FUNCTION_BLOCK AI_Temperature_Channel IMPLEMENTS I_AI_Temperature, I_AI_percentage
VAR_INPUT
	terminal_address		: WORD;
	CoE_communication_handler	: I_CoE_communication_handler;
END_VAR
VAR_OUTPUT
END_VAR
VAR
	_adc_min        : INT;
    _adc_max        : INT;
	_physical_min 	: INT;
	_physical_max 	: INT;
	_channel_number : UINT;
	_rValue			: REAL;
	_wcState		: BOOL;
	
	// ===============================================================================
	// CoE handling  
    // ==============
    _CoE_prop_handler      : CoE_property_handler;
    _CoE_channel_offset     : INT;
    index_1 				: WORD:= 16#8000 + INT_TO_WORD(_CoE_channel_offset);	
    // ====  CoE properties  ===========
	_p_Enable_user_scale    		: CoE_property(Index:=index_1 , SubIndex:=1, PropertyType:=Tc2_Utilities.ARGTYPE_BOOL, writable:=TRUE, propertyType:=0, pollingInterval:=T#5S);
	_p_Presentation 				: CoE_property(Index:=index_1 , SubIndex:=2, PropertyType:=Tc2_Utilities.ARGTYPE_USINT, writable:=TRUE, propertyType:=0, pollingInterval:=T#5S);			// DT0800EN03
	_p_Watchdog 					: CoE_property(Index:=index_1 , SubIndex:=5, PropertyType:=Tc2_Utilities.ARGTYPE_USINT, writable:=TRUE, propertyType:=0, pollingInterval:=T#5S);			// DT0801EN02
	_p_Enable_user_calibration  	: CoE_property(Index:=index_1 , SubIndex:=7, PropertyType:=Tc2_Utilities.ARGTYPE_BOOL, writable:=TRUE, propertyType:=0, pollingInterval:=T#5S);
	_p_Enable_vendor_calibration    : CoE_property(Index:=index_1 , SubIndex:=8, PropertyType:=Tc2_Utilities.ARGTYPE_BOOL, writable:=TRUE, propertyType:=0, pollingInterval:=T#5S);
	_p_Offset   					: CoE_property(Index:=index_1 , SubIndex:=17, PropertyType:=Tc2_Utilities.ARGTYPE_INT, writable:=TRUE, propertyType:=0, pollingInterval:=T#5S);
	_p_Gain 						: CoE_property(Index:=index_1 , SubIndex:=18, PropertyType:=Tc2_Utilities.ARGTYPE_DINT, writable:=TRUE, propertyType:=0, pollingInterval:=T#5S);
	_p_Default_output   			: CoE_property(Index:=index_1 , SubIndex:=19, PropertyType:=Tc2_Utilities.ARGTYPE_INT, writable:=TRUE, propertyType:=0, pollingInterval:=T#5S);
	_p_Default_output_ramp  		: CoE_property(Index:=index_1 , SubIndex:=20, PropertyType:=Tc2_Utilities.ARGTYPE_UINT, writable:=TRUE, propertyType:=0, pollingInterval:=T#5S);
	_p_User_calibration_offset  	: CoE_property(Index:=index_1 , SubIndex:=21, PropertyType:=Tc2_Utilities.ARGTYPE_INT, writable:=TRUE, propertyType:=0, pollingInterval:=T#5S);
	_p_User_calibration_gain    	: CoE_property(Index:=index_1 , SubIndex:=22, PropertyType:=Tc2_Utilities.ARGTYPE_UINT, writable:=TRUE, propertyType:=0, pollingInterval:=T#5S);
	// ==============
	_properties  : ARRAY[1..11]OF I_CoE_property:=[
		_p_Enable_user_scale, _p_Presentation, _p_Watchdog, _p_Enable_user_calibration, _p_Enable_vendor_calibration, _p_Offset,
		_p_Gain, _p_Default_output, _p_Default_output_ramp, _p_User_calibration_offset, _p_User_calibration_gain];
	// ===============================================================================
    
	
	//  ====  I_AI_percentage  ====
	_max_value 	: REAL:=10.0;
	_min_value 	: REAL:=0.0;
	_value: REAL;
	
	_errId: HAL_ErrorEnum;
    neg_wcState: f_trig;
END_VAR

// CoE Property handling 
_CoE_prop_handler(terminal_address:=terminal_address, CoE_communication_handler:=CoE_communication_handler, CoE_properties:=_properties);

neg_wcState(CLK:=_wcState);
IF neg_wcState.Q THEN
    ;
END_IF

PROPERTY errId : HAL_ErrorEnum
GET
errId := _errId;
END_GET
END_PROPERTY

METHOD FB_init : BOOL
VAR_INPUT
	bInitRetains 	: BOOL; // if TRUE, the retain variables are initialized (warm start / cold start)
	bInCopyCode 	: BOOL;  // if TRUE, the instance afterwards gets moved into the copy code (online change)
    adc_min         : INT;
    adc_max         : INT;
	physical_min 	: INT;
	physical_max 	: INT;
	channel_number  : UINT;
END_VAR

VAR
	i: UINT;
END_VAR

_adc_min        := adc_min;
_adc_max        := adc_max;
_physical_min 	:= physical_min;
_physical_max 	:= physical_max;
_channel_number :=channel_number;

CASE channel_number OF
	1:
		_CoE_channel_offset:=16#0;
	2:
		_CoE_channel_offset:=16#10;
	3:
		_CoE_channel_offset:=16#20;
	4:
		_CoE_channel_offset:=16#30;
END_CASE
END_METHOD

METHOD get_Default_output : BOOL
VAR
    targ_value : Tc2_Utilities.T_Arg;
END_VAR
VAR_OUTPUT
	value	: INT;
END_VAR
get_Default_output:=_p_Default_output.get_value(value=>targ_value, errId => );
IF get_Default_output THEN
    MEMCPY(ADR(value), targ_value.pData, targ_value.cbLen);
END_IF
END_METHOD

METHOD get_Default_output_ramp : BOOL
VAR
    targ_value : Tc2_Utilities.T_Arg;
END_VAR
VAR_OUTPUT
	value	: UINT;
END_VAR
get_Default_output_ramp:=_p_Default_output_ramp.get_value(value=>targ_value, errId => );
IF get_Default_output_ramp THEN
    MEMCPY(ADR(value), targ_value.pData, targ_value.cbLen);
END_IF
END_METHOD

METHOD get_Enable_user_calibration : BOOL
VAR
    targ_value : Tc2_Utilities.T_Arg;
END_VAR
VAR_OUTPUT
	value	: BOOL;
END_VAR
get_Enable_user_calibration:=_p_Enable_user_calibration.get_value(value=>targ_value, errId => );
IF get_Enable_user_calibration THEN
    MEMCPY(ADR(value), targ_value.pData, targ_value.cbLen);
END_IF
END_METHOD

METHOD get_Enable_user_scale : BOOL
VAR
    targ_value : Tc2_Utilities.T_Arg;
END_VAR
VAR_OUTPUT
	value	: BOOL;
END_VAR
get_Enable_user_scale:=_p_Enable_user_scale.get_value(value=>targ_value, errId => );
IF get_Enable_user_scale THEN
    MEMCPY(ADR(value), targ_value.pData, targ_value.cbLen);
END_IF
END_METHOD

METHOD get_Enable_vendor_calibration : BOOL
VAR
    targ_value : Tc2_Utilities.T_Arg;
END_VAR
VAR_OUTPUT
	value	: BOOL;
END_VAR
get_Enable_vendor_calibration:=_p_Enable_vendor_calibration.get_value(value=>targ_value, errId => );
IF get_Enable_vendor_calibration THEN
    MEMCPY(ADR(value), targ_value.pData, targ_value.cbLen);
END_IF
END_METHOD

METHOD get_Gain : BOOL
VAR
    targ_value : Tc2_Utilities.T_Arg;
END_VAR
VAR_OUTPUT
	value	: DINT;
END_VAR
get_Gain:=_p_Gain.get_value(value=>targ_value, errId => );
IF get_Gain THEN
    MEMCPY(ADR(value), targ_value.pData, targ_value.cbLen);
END_IF
END_METHOD

METHOD get_Offset : BOOL
VAR
    targ_value : Tc2_Utilities.T_Arg;
END_VAR
VAR_OUTPUT
	value	: INT;
END_VAR
get_Offset:=_p_Offset.get_value(value=>targ_value, errId => );
IF get_Offset THEN
    MEMCPY(ADR(value), targ_value.pData, targ_value.cbLen);
END_IF
END_METHOD

METHOD get_Presentation : BOOL
VAR
	usint_value: USINT;
    targ_value : Tc2_Utilities.T_Arg;
END_VAR
VAR_OUTPUT
	value	: ENU_DT0801EN03;
END_VAR
get_Presentation:=_p_Presentation.get_value(value=>targ_value, errId => );
IF get_Presentation THEN
    MEMCPY(ADR(usint_value), targ_value.pData, targ_value.cbLen);
    value:=USINT_TO_INT(usint_value);
END_IF
END_METHOD

METHOD get_User_calibration_gain : BOOL
VAR
    targ_value : Tc2_Utilities.T_Arg;
END_VAR
VAR_OUTPUT
	value	: UINT;
END_VAR
get_User_calibration_gain:=_p_User_calibration_gain.get_value(value=>targ_value, errId => );
IF get_User_calibration_gain THEN
    MEMCPY(ADR(value), targ_value.pData, targ_value.cbLen);
END_IF
END_METHOD

METHOD get_User_calibration_offset : BOOL
VAR
    targ_value : Tc2_Utilities.T_Arg;
END_VAR
VAR_OUTPUT
	value	: INT;
END_VAR
get_User_calibration_offset:=_p_User_calibration_offset.get_value(value=>targ_value, errId => );
IF get_User_calibration_offset THEN
    MEMCPY(ADR(value), targ_value.pData, targ_value.cbLen);
END_IF
END_METHOD

METHOD get_Watchdog : BOOL
VAR
	usint_value: USINT;
    targ_value : Tc2_Utilities.T_Arg;
END_VAR
VAR_OUTPUT
	value	: ENU_DT0800EN02;
END_VAR
get_Watchdog:=_p_Watchdog.get_value(value=>targ_value, errId => );
IF get_Watchdog THEN
    MEMCPY(ADR(usint_value), targ_value.pData, targ_value.cbLen);
    value:=USINT_TO_INT(usint_value);
END_IF
END_METHOD

PROPERTY io_status_Error : bool
GET
END_GET
SET
END_SET
END_PROPERTY

PROPERTY io_status_Limit_1_greater_value : bool
GET
END_GET
SET
END_SET
END_PROPERTY

PROPERTY io_status_Limit_1_smaller_value : bool
GET
END_GET
SET
END_SET
END_PROPERTY

PROPERTY io_status_Limit_2_greater_value : bool
GET
END_GET
SET
END_SET
END_PROPERTY

PROPERTY io_status_Limit_2_smaller_value : bool
GET
END_GET
SET
END_SET
END_PROPERTY

PROPERTY io_status_Overrange : bool
GET
END_GET
SET
END_SET
END_PROPERTY

PROPERTY io_status_Sync_error : bool
GET
END_GET
SET
END_SET
END_PROPERTY

PROPERTY io_status_TxPDO_State : bool
GET
END_GET
SET
END_SET
END_PROPERTY

PROPERTY io_status_TxPDO_Toggle : bool
GET
END_GET
SET
END_SET
END_PROPERTY

PROPERTY io_status_Underrange : bool
GET
END_GET
SET
END_SET
END_PROPERTY

PROPERTY max_value : REAL
GET
max_value := _max_value;
END_GET
SET
IF max_value <= 0 THEN
	_max_value := 0.0001;
ELSE
	_max_value := max_value;
END_IF
END_SET
END_PROPERTY

PROPERTY min_value : REAL
GET
min_value := _min_value;
END_GET
SET
_min_value := min_value;
END_SET
END_PROPERTY

PROPERTY rValue : REAL
GET
rValue:=_rValue;
END_GET
SET
IF rValue < DINT_TO_REAL(_physical_min) THEN
	_errId := 6;
ELSIF rValue > DINT_TO_REAL(_physical_max) THEN
	_errId := 7;
ELSE
	_rValue := rValue;
END_IF
END_SET
END_PROPERTY

METHOD set_Default_output : BOOL
VAR_INPUT
	value	: INT;
END_VAR
set_Default_output:=_p_Default_output.set_value(value:=Tc2_Utilities.F_INT(in:=value));
END_METHOD

METHOD set_Default_output_ramp : BOOL
VAR_INPUT
	value	: UINT;
END_VAR
set_Default_output_ramp:=_p_Default_output_ramp.set_value(value:=Tc2_Utilities.F_UINT(in:=value));
END_METHOD

METHOD set_Enable_user_calibration : BOOL
VAR_INPUT
	value	: BOOL;
END_VAR
set_Enable_user_calibration:=_p_Enable_user_calibration.set_value(value:=Tc2_Utilities.F_BOOL(in:=value));
END_METHOD

METHOD set_Enable_user_scale : BOOL
VAR_INPUT
	value	: BOOL;
END_VAR
set_Enable_user_scale:=_p_Enable_user_scale.set_value(value:=Tc2_Utilities.F_BOOL(in:=value));
END_METHOD

METHOD set_Enable_vendor_calibration : BOOL
VAR_INPUT
	value	: BOOL;
END_VAR
set_Enable_vendor_calibration:=_p_Enable_vendor_calibration.set_value(value:=Tc2_Utilities.F_BOOL(in:=value));
END_METHOD

METHOD set_Gain : BOOL
VAR_INPUT
	value	: DINT;
END_VAR
set_Gain:=_p_Gain.set_value(value:=Tc2_Utilities.F_DINT(in:=value));
END_METHOD

METHOD set_Offset : BOOL
VAR_INPUT
	value	: INT;
END_VAR
set_Offset:=_p_Offset.set_value(value:=Tc2_Utilities.F_INT(in:=value));
END_METHOD

METHOD set_Presentation : BOOL
VAR_INPUT
	value	: ENU_DT0801EN03;
END_VAR
set_Presentation:=_p_Presentation.set_value(value:=Tc2_Utilities.F_USINT(in:=INT_TO_USINT(value)));
END_METHOD

METHOD set_User_calibration_gain : BOOL
VAR_INPUT
	value	: UINT;
END_VAR
set_User_calibration_gain:=_p_User_calibration_gain.set_value(value:=Tc2_Utilities.F_UINT(in:=value));
END_METHOD

METHOD set_User_calibration_offset : BOOL
VAR_INPUT
	value	: INT;
END_VAR
set_User_calibration_offset:=_p_User_calibration_offset.set_value(value:=Tc2_Utilities.F_INT(in:=value));
END_METHOD

METHOD set_Watchdog : BOOL
VAR_INPUT
	value	: ENU_DT0800EN02;
END_VAR
set_Watchdog:=_p_Watchdog.set_value(value:=Tc2_Utilities.F_USINT(in:=INT_TO_USINT(value)));
END_METHOD

PROPERTY terminal_value : int
SET
linear_adc_to_phy(
	physical_min	:= _physical_min, 
	physical_max	:= _physical_max, 
	adc_min			:= _adc_min, 
	adc_max			:= _adc_max, 
	adc_value		:= terminal_value, 
	physical_value	=> _rValue, 
	errId			=> _errId
);

linear_adc_to_phy(
	physical_min	:= 0, 
	physical_max	:= 100, 
	adc_min			:= REAL_TO_DINT(_min_value), 
	adc_max			:= REAL_TO_DINT(_max_value), 
	adc_value		:= REAL_TO_DINT(_rValue), 
	physical_value	=> _value, 
	errId			=> _errId
);
END_SET
END_PROPERTY

PROPERTY value : REAL
GET
value := _value;
END_GET
END_PROPERTY

PROPERTY wcState : bool
GET
wcState:=_wcState;
END_GET
SET
_wcState:=wcState;
END_SET
END_PROPERTY

END_FUNCTION_BLOCK

(* stored: Version 1.1.0.1, ProductVersion 3.1.4024.9
   POU AI_Temperature_Channel: Id {6bbe721b-eb3d-04ba-01ae-2009e4a41bd1}, SpecialFunc None
   Folder config: Id {bb2195d8-7083-08cc-32cb-38091d042fe0}
   Folder HAL: Id {6c0feffb-c4d0-0d64-1a03-4b31aee82e86}
   Folder IO: Id {3507ca37-d29f-093d-3619-545f2b15d211}
   Property errId: Id {30eadb91-2fc6-03c4-3e0c-22123c9f8a94}
   Get Get: Id {89495df1-107f-02e7-3f39-5c962767d6e1}
   Method FB_init: Id {922758f3-0b9f-0c30-218f-0a42385c584d}
   Method get_Default_output: Id {7427f853-14c9-0a2e-2baa-c4fa4c9b0918}
   Method get_Default_output_ramp: Id {fac8043d-224a-046c-3bc5-7ccc20cb6905}
   Method get_Enable_user_calibration: Id {253a4690-52c4-0a69-1f9e-fd2e16030921}
   Method get_Enable_user_scale: Id {c8577104-d830-03d1-3d11-85cfcfe93a61}
   Method get_Enable_vendor_calibration: Id {f1657459-6fc9-0987-363b-f57e47b889b2}
   Method get_Gain: Id {0378892b-0be5-0128-151d-c53069676214}
   Method get_Offset: Id {875fb64f-aa95-0b6c-18b9-f83d0a09f168}
   Method get_Presentation: Id {013ad0f9-4b38-06b8-2755-04279490b138}
   Method get_User_calibration_gain: Id {48d2e637-48d9-0313-0747-ae61d5d29f7c}
   Method get_User_calibration_offset: Id {32dbbe99-4b0f-0c99-3cc8-ede93d249979}
   Method get_Watchdog: Id {b8075401-7e9f-060b-3ed1-949acdcf1937}
   Property io_status_Error: Id {b301b5fa-842b-0581-1acf-871c72bcc9ae}
   Get Get: Id {f41f8146-8cd1-0b51-18cf-30f4c7059e51}
   Set Set: Id {ff93eaca-5456-0de1-1a93-4e7d8ca568ec}
   Property io_status_Limit_1_greater_value: Id {cb696e6a-0e97-001d-26b9-34533094c579}
   Get Get: Id {65dbc163-02cd-0043-131c-4bf4e5d6aee8}
   Set Set: Id {b9ec8874-a90d-0ced-1805-d747f575c6ee}
   Property io_status_Limit_1_smaller_value: Id {c981e412-e11d-0d11-3778-9d82e4e97f33}
   Get Get: Id {a2b858c9-26bf-05c7-1b1d-28ac79eb9b14}
   Set Set: Id {afe2d63b-cb6d-055d-169f-6abd4953db83}
   Property io_status_Limit_2_greater_value: Id {0327c59f-eba8-09df-244f-99c5a7c56ec5}
   Get Get: Id {9f94b768-bbfd-0169-2eb6-45ee37b304fb}
   Set Set: Id {a77150a2-3e78-051b-2513-d0c987742a25}
   Property io_status_Limit_2_smaller_value: Id {8558f92e-10be-0652-30b4-2f7d5ecabbb0}
   Get Get: Id {29f65031-684e-02da-0af4-8485e4f44869}
   Set Set: Id {a1a1ad77-c1b2-0843-084f-933b1fb4411f}
   Property io_status_Overrange: Id {a7432bc9-fe33-051d-27b7-5108bd7fa008}
   Get Get: Id {b7e93c44-5d3f-09a7-338f-2fc8b07ede3e}
   Set Set: Id {324e2887-2d21-0344-3038-b2f145d66248}
   Property io_status_Sync_error: Id {6a9fcfb3-ac71-09d4-0a1d-90c8f350fab0}
   Get Get: Id {86825138-291c-019a-3724-49a74208cee6}
   Set Set: Id {c33cd3ca-780c-0937-1e38-67680fd5128b}
   Property io_status_TxPDO_State: Id {45c99470-3221-042b-0ccc-0d0e2f9a0fb7}
   Get Get: Id {1b358420-7941-0aca-3d0c-cf34ba599ddb}
   Set Set: Id {320448fc-9043-09b1-0911-686536b38603}
   Property io_status_TxPDO_Toggle: Id {f0c72f6c-ab77-0e01-3056-dea2d31d5105}
   Get Get: Id {3b6bbf86-c457-025f-2a65-47ed72327b47}
   Set Set: Id {25f115a3-c71e-078a-360a-ee19b1d7fe5e}
   Property io_status_Underrange: Id {545964b2-4f8e-0ac8-239f-be6b9b1aeb83}
   Get Get: Id {8035c8a8-e3d5-075b-1335-0a3918e7da58}
   Set Set: Id {8786be1a-f7d7-0670-30e7-72ec09619d56}
   Property max_value: Id {41924a96-b9bb-06f3-2986-05878bd58d97}
   Get Get: Id {9ed71e7f-2071-0687-1504-44d3f0f7bc0a}
   Set Set: Id {98876934-9793-0b65-1258-874be1423bce}
   Property min_value: Id {75265f7f-1c0a-09c6-14d2-ff3db43460d6}
   Get Get: Id {44a260da-2638-0d4d-37bd-c205aaa17587}
   Set Set: Id {355c3a65-f520-0f98-2458-4e7ec12585e0}
   Property rValue: Id {0ef95a23-2848-052e-1f94-5118a5eab3bc}
   Get Get: Id {6586983f-bec8-0b4e-0f34-dfafb3f79d78}
   Set Set: Id {7ce133b4-5134-0008-1aae-4a0494bd588e}
   Method set_Default_output: Id {80e2a255-8654-03c1-0a95-90ae41b7d10a}
   Method set_Default_output_ramp: Id {4f5bf14a-46c9-0f57-28ab-832af1aec365}
   Method set_Enable_user_calibration: Id {f42a704b-c420-0d63-0a2d-3e58b804b97a}
   Method set_Enable_user_scale: Id {096c7aef-c307-0e2f-0f2a-19c7ac4a4165}
   Method set_Enable_vendor_calibration: Id {c2dcebc2-8e9a-0dd7-1092-05ac0efba035}
   Method set_Gain: Id {de30f028-a28e-0126-12a8-0fab9b34f94a}
   Method set_Offset: Id {80eca5c9-6ae1-0a49-193a-2c332611c617}
   Method set_Presentation: Id {5a20384b-dff8-06aa-3c3e-1fc798c4c674}
   Method set_User_calibration_gain: Id {81ae2f78-c6a2-0462-1bbc-8e57925e4f97}
   Method set_User_calibration_offset: Id {7b2fe8ba-0327-04a5-1711-d0f89c395523}
   Method set_Watchdog: Id {a58f1101-5e77-0090-1b75-82d4f86d3414}
   Property terminal_value: Id {967080f2-c801-0524-0a1d-95eb8af69e09}
   Set Set: Id {cd92f733-70c4-0b4a-090c-3157f4ede09e}
   Property value: Id {4018688d-f092-0037-20fb-77031041f7a5}
   Get Get: Id {b27b22ad-23da-0676-0121-1b7f9afff176}
   Property wcState: Id {049b3df0-6b4d-012d-2d34-772f314d1142}
   Get Get: Id {43e4ad3b-fbdc-008b-148b-6ae6f331fb44}
   Set Set: Id {496749e1-9e1a-00f0-0aa0-4f167c0e5976} *)
